(* Schneider Machine Expert - Basic project Test_Conveyor, file version 3.0.0.0 *)
(* ProjectInformations: Name=Test_Conveyor *)

HARDWARE
  Cpu 0: TM221C24R
  SerialLineConfiguration: Baud=Baud19200, Parity=ParityEven, DataBits=DataBits8, StopBits=StopBits1, PhysicalMedium=PhysicalMediumRs485, TransmissionMode=TransmissionModeModbusRtu, SlaveId=1, Addressing=SlaveAddressing
  MastTask: UsePeriodScanMode=false, PeriodScan=100
  FastTask: Period=255
  CpuBehavior: StartingMode=StartAsPreviousState, AutoSaveRamOnEeprom=true, WatchdogPeriod=250

SYMBOLS  (address, symbol, comment, settings)
  %M0       CONV_RUN  "Conveyor Running"
  %I0.0     PB_START
  %I0.1     PB_STOP
  %I0.2     SENS1
  %I0.3     SENS2
  %Q0.0     CONV_MTR
  %Q0.1     LT_STA1
  %Q0.2     LT_STA2

POU Test_Conveyor
  (* SectionNumber=1 *)

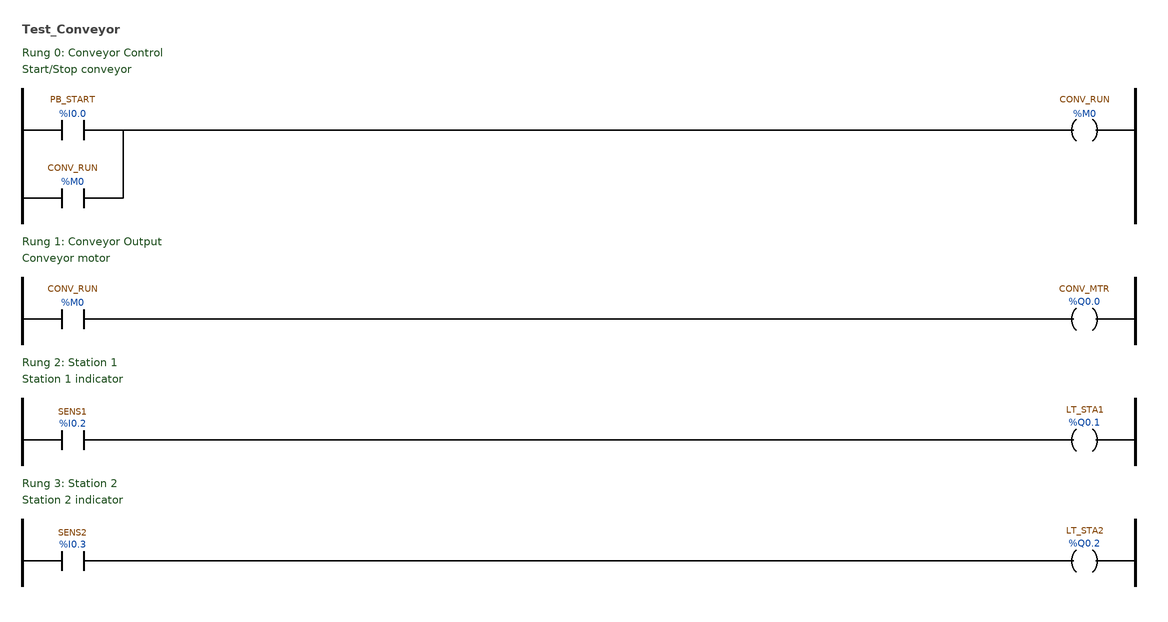

// Rung 0: Conveyor Control
// Start/Stop conveyor
  LD %I0.0                (* PB_START *)
  OR %M0                  (* CONV_RUN *)
  ST %M0                  (* CONV_RUN *)
  // as ST:
  //   CONV_RUN := PB_START OR CONV_RUN;

// Rung 1: Conveyor Output
// Conveyor motor
  LD %M0                  (* CONV_RUN *)
  ST %Q0.0                (* CONV_MTR *)
  // as ST:
  //   CONV_MTR := CONV_RUN;

// Rung 2: Station 1
// Station 1 indicator
  LD %I0.2                (* SENS1 *)
  ST %Q0.1                (* LT_STA1 *)
  // as ST:
  //   LT_STA1 := SENS1;

// Rung 3: Station 2
// Station 2 indicator
  LD %I0.3                (* SENS2 *)
  ST %Q0.2                (* LT_STA2 *)
  // as ST:
  //   LT_STA2 := SENS2;
